{attribute addProperty BoxType "EP2339-0042-0018"}
{attribute addProperty Id "DI_X01AT %I*ARRAY[0..1] OF DI_X_E4AEF59E429496728842949672950DI_X02AT %I*ARRAY[0..1] OF DI_X_E4AEF59E429496728842949672950DI_X03AT %I*ARRAY[0..1] OF DI_X_E4AEF59E429496728842949672950DI_X04AT %I*ARRAY[0..1] OF DI_X_E4AEF59E429496728842949672950DI_X05AT %I*ARRAY[0..1] OF DI_X_E4AEF59E429496728842949672950DI_X06AT %I*ARRAY[0..1] OF DI_X_E4AEF59E429496728842949672950DI_X07AT %I*ARRAY[0..1] OF DI_X_E4AEF59E429496728842949672950DI_X08AT %I*ARRAY[0..1] OF DI_X_E4AEF59E429496728842949672950DO_X01AT %Q*ARRAY[0..1] OF DO_X_7F374EB0429496728842949672950DO_X02AT %Q*ARRAY[0..1] OF DO_X_7F374EB0429496728842949672950DO_X03AT %Q*ARRAY[0..1] OF DO_X_7F374EB0429496728842949672950DO_X04AT %Q*ARRAY[0..1] OF DO_X_7F374EB0429496728842949672950DO_X05AT %Q*ARRAY[0..1] OF DO_X_7F374EB0429496728842949672950DO_X06AT %Q*ARRAY[0..1] OF DO_X_7F374EB0429496728842949672950DO_X07AT %Q*ARRAY[0..1] OF DO_X_7F374EB0429496728842949672950DO_X08AT %Q*ARRAY[0..1] OF DO_X_7F374EB0429496728842949672950WcStateAT %I*WcState_F855686C1620InfoDataAT %I*InfoData_192954DE1620"}
{attribute addProperty CRC "1601622921"}
{attribute addProperty SizeInBites "4294967200"}
{attribute addProperty SizeInBytes "68719476724"}
TYPE EP2339_1E71110B :
STRUCT
	{attribute addProperty Name "DI_X01"}
	DI_X01 : ARRAY[0..1] OF DI_X_E4AEF59E;
	{attribute addProperty Name "DI_X02"}
	DI_X02 : ARRAY[0..1] OF DI_X_E4AEF59E;
	{attribute addProperty Name "DI_X03"}
	DI_X03 : ARRAY[0..1] OF DI_X_E4AEF59E;
	{attribute addProperty Name "DI_X04"}
	DI_X04 : ARRAY[0..1] OF DI_X_E4AEF59E;
	{attribute addProperty Name "DI_X05"}
	DI_X05 : ARRAY[0..1] OF DI_X_E4AEF59E;
	{attribute addProperty Name "DI_X06"}
	DI_X06 : ARRAY[0..1] OF DI_X_E4AEF59E;
	{attribute addProperty Name "DI_X07"}
	DI_X07 : ARRAY[0..1] OF DI_X_E4AEF59E;
	{attribute addProperty Name "DI_X08"}
	DI_X08 : ARRAY[0..1] OF DI_X_E4AEF59E;
	{attribute addProperty Name "DO_X01"}
	DO_X01 : ARRAY[0..1] OF DO_X_7F374EB0;
	{attribute addProperty Name "DO_X02"}
	DO_X02 : ARRAY[0..1] OF DO_X_7F374EB0;
	{attribute addProperty Name "DO_X03"}
	DO_X03 : ARRAY[0..1] OF DO_X_7F374EB0;
	{attribute addProperty Name "DO_X04"}
	DO_X04 : ARRAY[0..1] OF DO_X_7F374EB0;
	{attribute addProperty Name "DO_X05"}
	DO_X05 : ARRAY[0..1] OF DO_X_7F374EB0;
	{attribute addProperty Name "DO_X06"}
	DO_X06 : ARRAY[0..1] OF DO_X_7F374EB0;
	{attribute addProperty Name "DO_X07"}
	DO_X07 : ARRAY[0..1] OF DO_X_7F374EB0;
	{attribute addProperty Name "DO_X08"}
	DO_X08 : ARRAY[0..1] OF DO_X_7F374EB0;
	{attribute addProperty Name "WcState"}
	WcState : WcState_F855686C;
	{attribute addProperty Name "InfoData"}
	InfoData : InfoData_192954DE;
END_STRUCT
END_TYPE

(* stored: Version 1.2.0.0, ProductVersion 3.1.4024.9
   DUT EP2339_1E71110B: Id {c8ca144a-38ca-4327-aecd-c4d5bae53e36} *)
